FUNCTION alg_a_TledQ2: BOOL
VAR_INPUT
    state: STATE;
END_VAR

alg_a_TledQ2 := (state.dvar_M_led2) = (elit_On);

END_FUNCTION

(* stored: ProductVersion 3.1.0.18, Version 1.1.0.1 *)
